{attribute 'call_after_init'}
FUNCTION_BLOCK FB_Laser_Test EXTENDS FB_TestSuite
VAR_INPUT
END_VAR
VAR_OUTPUT
END_VAR
VAR
END_VAR

RawVoltageScales1();
RawVoltageScales2();
RawVoltageScales3();
LowVoltageTriggersError();
ErrorLatches();
ErrorResets();
NoError();

METHOD ErrorLatches
VAR
	fbLaser : FB_Laser;
	stSetpoints : ST_LaserSetpoints;
END_VAR
TEST('ErrorLatches');

// Trigger low voltage error
fbLaser := F_Laser_Error(stSetpoints => stSetpoints);

// Give non-erronuous input. Laser should stary latched
fbLaser(bAmphosOn := FALSE, stSetpoints := stSetpoints);
AssertTrue(fbLaser.bError, 'Laser did not stay latched');

TEST_FINISHED();
END_METHOD

METHOD ErrorResets
VAR
	fbLaser : FB_Laser;
	stSetpoints : ST_LaserSetpoints;
END_VAR
TEST('ErrorResets');

fbLaser := F_Laser_Error(stSetpoints => stSetpoints);

// Resetting the error on the laser should unlatch the system
fbLaser.Reset();
fbLaser(bAmphosOn := FALSE, stSetpoints := stSetpoints);
AssertFalse(fbLaser.bError, 'System did not unlatch when reset');

TEST_FINISHED();
END_METHOD

METHOD LowVoltageTriggersError
VAR
	fbLaser : FB_Laser := F_Laser_Error();
END_VAR
TEST('LowVoltageErrorTriggers');

AssertTrue(fbLaser.bError, 'Error not triggered');

TEST_FINISHED();
END_METHOD

METHOD NoError
VAR
	fbLaser : FB_Laser;
	stSetpoints : ST_LaserSetpoints := F_LaserSetpoints();
END_VAR
TEST('NoError');

fbLaser(
	nVoltageRaw := 16#7736,
	bAmphosOn := TRUE,
	stSetpoints := stSetpoints
);
AssertFalse(fbLaser.bError, 'Error fasely detected');

TEST_FINISHED();
END_METHOD

METHOD RawVoltageScales1
VAR
	fbLaser : FB_Laser;
	stSetpoints : ST_LaserSetpoints := F_LaserSetpoints();
END_VAR
TEST('RawVoltageScales1');

fbLaser(nVoltageRaw := 16#0000, stSetpoints := stSetpoints);
AssertEquals_LREAL(0, fbLaser.fVoltage, 0.01, 'Incorrect voltage scaling');

TEST_FINISHED();
END_METHOD

METHOD RawVoltageScales2
VAR
	fbLaser : FB_Laser;
	stSetpoints : ST_LaserSetpoints := F_LaserSetpoints();
END_VAR
TEST('RawVoltageScales2');

fbLaser(nVoltageRaw := 16#7736, stSetpoints := stSetpoints);
AssertEquals_LREAL(10, fbLaser.fVoltage, 0.01, 'Incorrect Amphos voltage scaling');

TEST_FINISHED();
END_METHOD

METHOD RawVoltageScales3
VAR
	fbLaser : FB_Laser;
	stSetpoints : ST_LaserSetpoints := F_LaserSetpoints();
END_VAR
TEST('RawVoltageScales3');

// Test behavior when given an overrange raw input
fbLaser(nVoltageRaw := 16#7FFF, stSetpoints := stSetpoints);
AssertEquals_LREAL(10, fbLaser.fVoltage, 0.01, 'Incorrect Amphos voltage scaling');

TEST_FINISHED();
END_METHOD

END_FUNCTION_BLOCK

(* stored: Version 1.1.0.1, ProductVersion 3.1.4020.14
   POU FB_Laser_Test: Id {860a4e36-c631-4b10-9868-fa916183422c}, SpecialFunc None
   Method ErrorLatches: Id {321319df-1a26-4143-9715-3e98483394c1}
   Method ErrorResets: Id {efd0dfe7-adcc-4695-afec-ce88fa7bc915}
   Method LowVoltageTriggersError: Id {e4a76605-25ac-44af-b6eb-ae4e39c6c5fc}
   Method NoError: Id {beb067e4-00b8-4802-9bf4-953e8a2f2d30}
   Method RawVoltageScales1: Id {7c1b2d03-d119-496c-83e5-1c9d35970c07}
   Method RawVoltageScales2: Id {2f28fb45-46b6-492d-b115-bd95d8cb3d85}
   Method RawVoltageScales3: Id {f2882aba-46b2-48e9-8e57-313ab9044dae} *)
